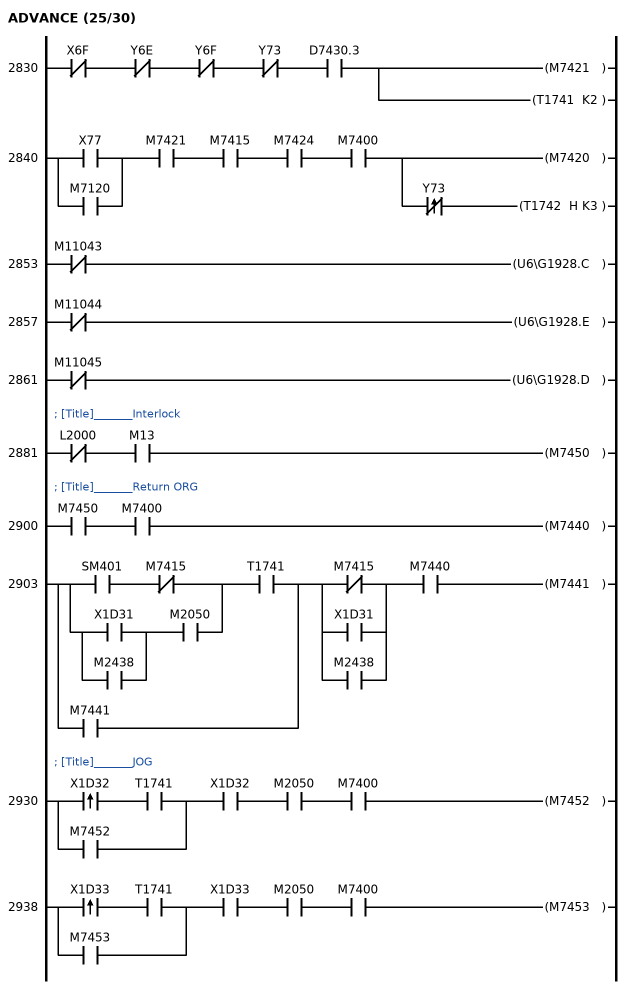
[picture p384: ladder of ADVANCE, rungs at steps 2830 to 2938]
2830  LDI     X6F
      ANI     Y6E
      ANI     Y6F
      ANI     Y73
      AND     D7430.3
      OUT     M7421
      OUT     T1741 K2
2840  LD      X77
      OR      M7120
      AND     M7421
      AND     M7415
      AND     M7424
      AND     M7400
      OUT     M7420
      ANDPI   Y73
      OUTH    T1742 K3
2853  LDI     M11043
      OUT     U6\G1928.C
2857  LDI     M11044
      OUT     U6\G1928.E
2861  LDI     M11045
      OUT     U6\G1928.D
; 
; [Title]_______Interlock
; 
2881  LDI     L2000
      AND     M13
      OUT     M7450
; 
; [Title]_______Return ORG
; 
2900  LD      M7450
      AND     M7400
      OUT     M7440
2903  LD      SM401
      ANI     M7415
      LD      X1D31
      OR      M2438
      AND     M2050
      ORB
      AND     T1741
      OR      M7441
      LDI     M7415
      OR      X1D31
      OR      M2438
      ANB
      AND     M7440
      OUT     M7441
; 
; [Title]_______JOG
; 
2930  LDP     X1D32
      AND     T1741
      OR      M7452
      AND     X1D32
      AND     M2050
      AND     M7400
      OUT     M7452
2938  LDP     X1D33
      AND     T1741
      OR      M7453
      AND     X1D33
      AND     M2050
      AND     M7400
      OUT     M7453
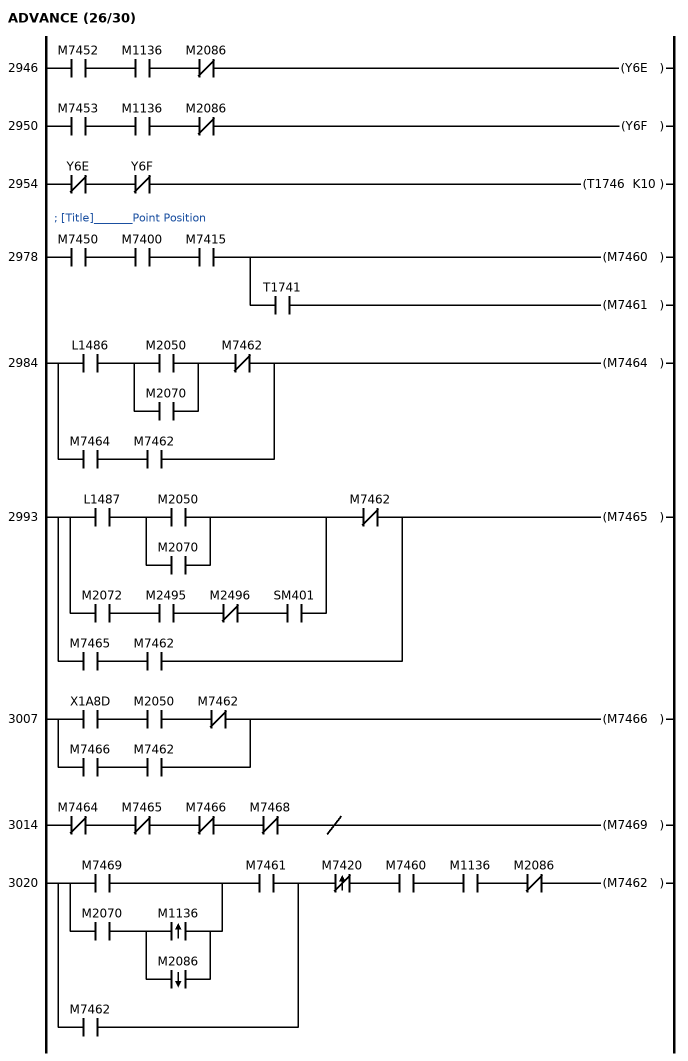
2946  LD      M7452
      AND     M1136
      ANI     M2086
      OUT     Y6E
2950  LD      M7453
      AND     M1136
      ANI     M2086
      OUT     Y6F
2954  LDI     Y6E
      ANI     Y6F
      OUT     T1746 K10
; 
; [Title]_______Point Position
; 
2978  LD      M7450
      AND     M7400
      AND     M7415
      OUT     M7460
      AND     T1741
      OUT     M7461
2984  LD      L1486
      LD      M2050
      OR      M2070
      ANB
      ANI     M7462
      LD      M7464
      AND     M7462
      ORB
      OUT     M7464
2993  LD      L1487
      LD      M2050
      OR      M2070
      ANB
      LD      M2072
      AND     M2495
      ANI     M2496
      AND     SM401
      ORB
      ANI     M7462
      LD      M7465
      AND     M7462
      ORB
      OUT     M7465
3007  LD      X1A8D
      AND     M2050
      ANI     M7462
      LD      M7466
      AND     M7462
      ORB
      OUT     M7466
3014  LDI     M7464
      ANI     M7465
      ANI     M7466
      ANI     M7468
      INV
      OUT     M7469
3020  LD      M7469
      LD      M2070
      LDP     M1136
      ORF     M2086
      ANB
      ORB
      AND     M7461
      OR      M7462
      ANDPI   M7420
      AND     M7460
      AND     M1136
      ANI     M2086
      OUT     M7462
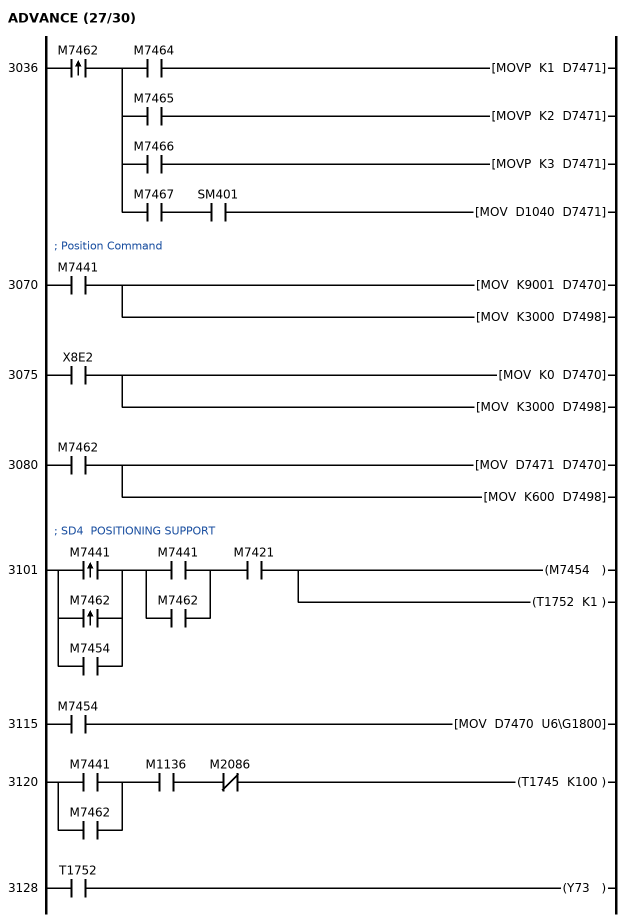
3036  LDP     M7462
      MPS
      AND     M7464
      MOVP    K1 D7471
      MRD
      AND     M7465
      MOVP    K2 D7471
      MRD
      AND     M7466
      MOVP    K3 D7471
      MPP
      AND     M7467
      AND     SM401
      MOV     D1040 D7471
; 
; Position Command
; 
3070  LD      M7441
      MOV     K9001 D7470
      MOV     K3000 D7498
3075  LD      X8E2
      MOV     K0 D7470
      MOV     K3000 D7498
3080  LD      M7462
      MOV     D7471 D7470
      MOV     K600 D7498
; 
; SD4  POSITIONING SUPPORT
; 
3101  LDP     M7441
      ORP     M7462
      OR      M7454
      LD      M7441
      OR      M7462
      ANB
      AND     M7421
      OUT     M7454
      OUT     T1752 K1
3115  LD      M7454
      MOV     D7470 U6\G1800
3120  LD      M7441
      OR      M7462
      AND     M1136
      ANI     M2086
      OUT     T1745 K100
3128  LD      T1752
      OUT     Y73
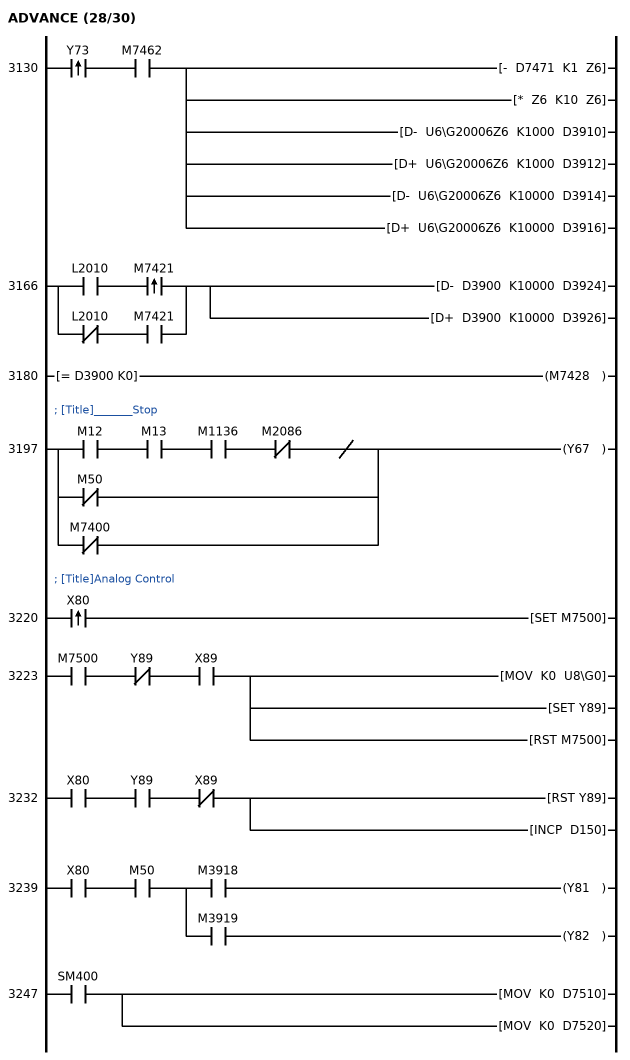
3130  LDP     Y73
      AND     M7462
      -       D7471 K1 Z6
      *       Z6 K10 Z6
      D-      U6\G20006Z6 K1000 D3910
      D+      U6\G20006Z6 K1000 D3912
      D-      U6\G20006Z6 K10000 D3914
      D+      U6\G20006Z6 K10000 D3916
3166  LD      L2010
      ANDP    M7421
      LDI     L2010
      AND     M7421
      ORB
      D-      D3900 K10000 D3924
      D+      D3900 K10000 D3926
3180  LD=     D3900 K0
      OUT     M7428
; 
; [Title]_______Stop
; 
3197  LD      M12
      AND     M13
      AND     M1136
      ANI     M2086
      INV
      ORI     M50
      ORI     M7400
      OUT     Y67
; 
; [Title]Analog Control
; 
3220  LDP     X80
      SET     M7500
3223  LD      M7500
      ANI     Y89
      AND     X89
      MOV     K0 U8\G0
      SET     Y89
      RST     M7500
3232  LD      X80
      AND     Y89
      ANI     X89
      RST     Y89
      INCP    D150
3239  LD      X80
      AND     M50
      MPS
      AND     M3918
      OUT     Y81
      MPP
      AND     M3919
      OUT     Y82
3247  LD      SM400
      MOV     K0 D7510
      MOV     K0 D7520
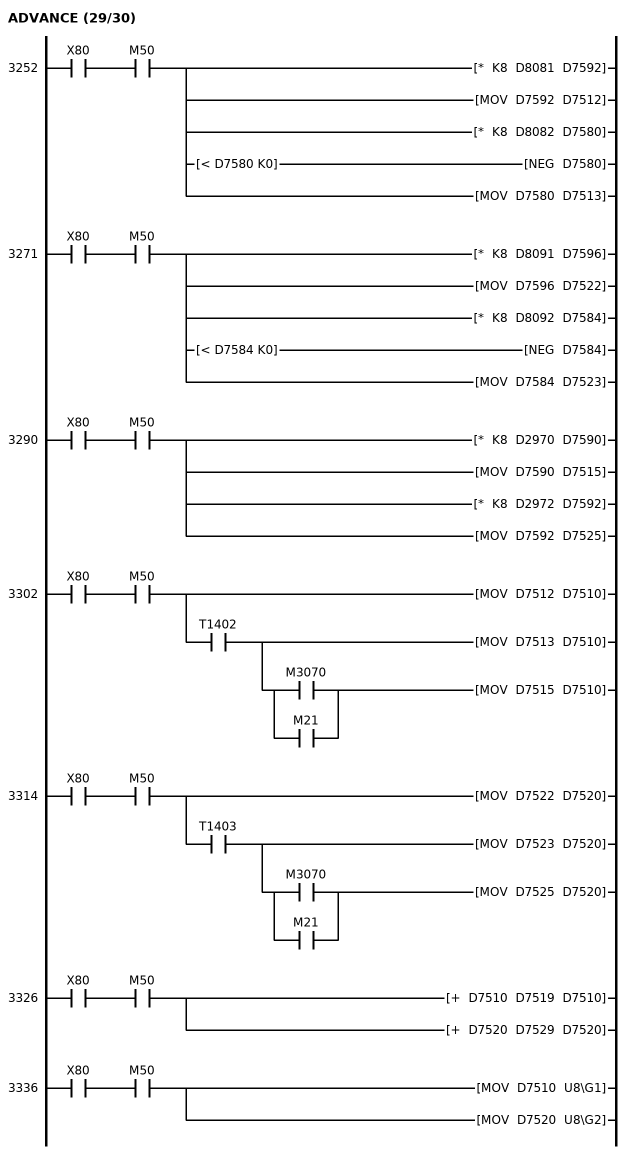
3252  LD      X80
      AND     M50
      *       K8 D8081 D7592
      MOV     D7592 D7512
      *       K8 D8082 D7580
      MPS
      AND<    D7580 K0
      NEG     D7580
      MPP
      MOV     D7580 D7513
3271  LD      X80
      AND     M50
      *       K8 D8091 D7596
      MOV     D7596 D7522
      *       K8 D8092 D7584
      MPS
      AND<    D7584 K0
      NEG     D7584
      MPP
      MOV     D7584 D7523
3290  LD      X80
      AND     M50
      *       K8 D2970 D7590
      MOV     D7590 D7515
      *       K8 D2972 D7592
      MOV     D7592 D7525
3302  LD      X80
      AND     M50
      MOV     D7512 D7510
      AND     T1402
      MOV     D7513 D7510
      LD      M3070
      OR      M21
      ANB
      MOV     D7515 D7510
3314  LD      X80
      AND     M50
      MOV     D7522 D7520
      AND     T1403
      MOV     D7523 D7520
      LD      M3070
      OR      M21
      ANB
      MOV     D7525 D7520
3326  LD      X80
      AND     M50
      +       D7510 D7519 D7510
      +       D7520 D7529 D7520
3336  LD      X80
      AND     M50
      MOV     D7510 U8\G1
      MOV     D7520 U8\G2
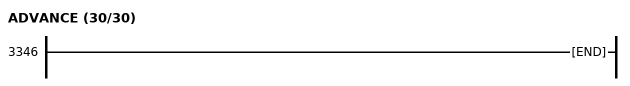
3346  END
END_PROGRAM

PROGRAM ALARM
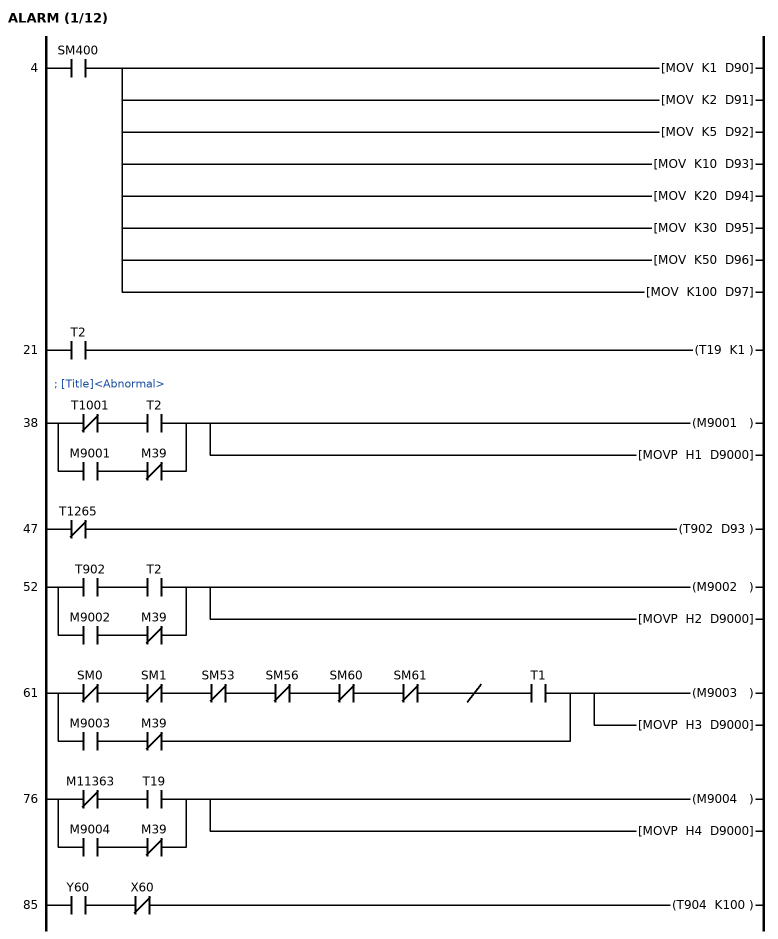
; 
; 
; 
4     LD      SM400
      MOV     K1 D90
      MOV     K2 D91
      MOV     K5 D92
      MOV     K10 D93
      MOV     K20 D94
      MOV     K30 D95
      MOV     K50 D96
      MOV     K100 D97
21    LD      T2
      OUT     T19 K1
; 
; [Title]<Abnormal>
38    LDI     T1001
      AND     T2
      LD      M9001
      ANI     M39
      ORB
      OUT     M9001
      MOVP    H1 D9000
47    LDI     T1265
      OUT     T902 D93
52    LD      T902
      AND     T2
      LD      M9002
      ANI     M39
      ORB
      OUT     M9002
      MOVP    H2 D9000
61    LDI     SM0
      ANI     SM1
      ANI     SM53
      ANI     SM56
      ANI     SM60
      ANI     SM61
      INV
      AND     T1
      LD      M9003
      ANI     M39
      ORB
      OUT     M9003
      MOVP    H3 D9000
76    LDI     M11363
      AND     T19
      LD      M9004
      ANI     M39
      ORB
      OUT     M9004
      MOVP    H4 D9000
85    LD      Y60
      ANI     X60
      OUT     T904 K100
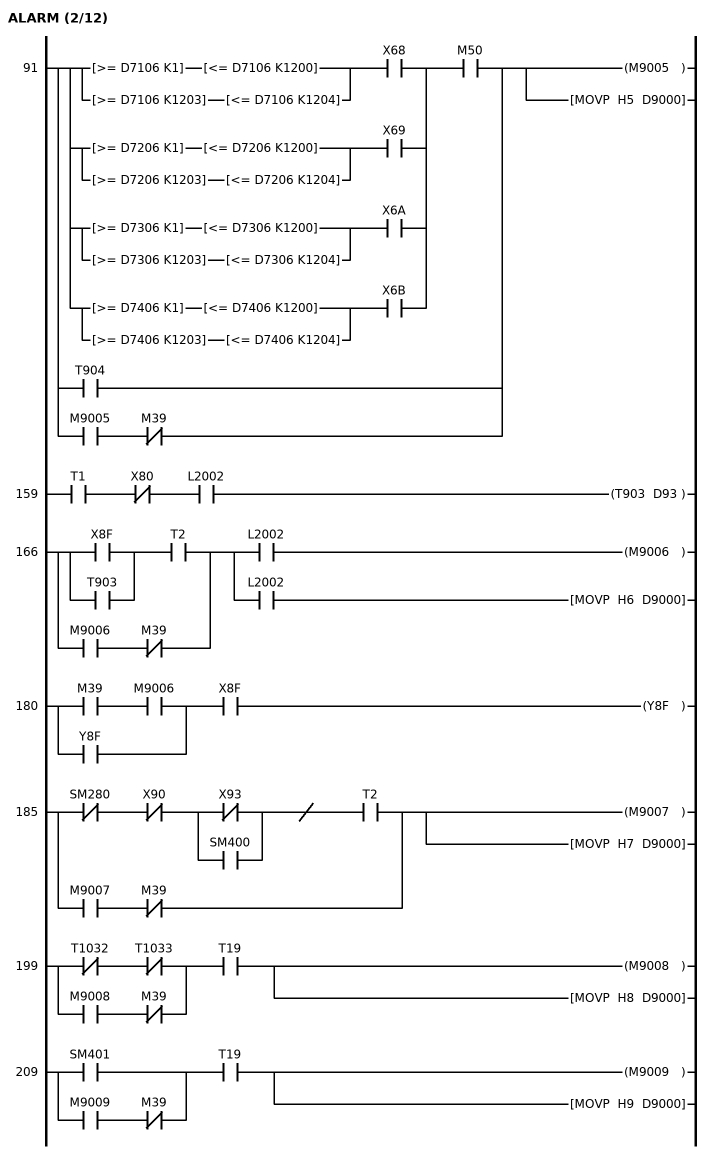
91    LD>=    D7106 K1
      AND<=   D7106 K1200
      LD>=    D7106 K1203
      AND<=   D7106 K1204
      ORB
      AND     X68
      LD>=    D7206 K1
      AND<=   D7206 K1200
      LD>=    D7206 K1203
      AND<=   D7206 K1204
      ORB
      AND     X69
      ORB
      LD>=    D7306 K1
      AND<=   D7306 K1200
      LD>=    D7306 K1203
      AND<=   D7306 K1204
      ORB
      AND     X6A
      ORB
      LD>=    D7406 K1
      AND<=   D7406 K1200
      LD>=    D7406 K1203
      AND<=   D7406 K1204
      ORB
      AND     X6B
      ORB
      AND     M50
      OR      T904
      LD      M9005
      ANI     M39
      ORB
      OUT     M9005
      MOVP    H5 D9000
159   LD      T1
      ANI     X80
      AND     L2002
      OUT     T903 D93
166   LD      X8F
      OR      T903
      AND     T2
      LD      M9006
      ANI     M39
      ORB
      MPS
      AND     L2002
      OUT     M9006
      MPP
      AND     L2002
      MOVP    H6 D9000
180   LD      M39
      AND     M9006
      OR      Y8F
      AND     X8F
      OUT     Y8F
185   LDI     SM280
      ANI     X90
      LDI     X93
      OR      SM400
      ANB
      INV
      AND     T2
      LD      M9007
      ANI     M39
      ORB
      OUT     M9007
      MOVP    H7 D9000
199   LDI     T1032
      ANI     T1033
      LD      M9008
      ANI     M39
      ORB
      AND     T19
      OUT     M9008
      MOVP    H8 D9000
209   LD      SM401
      LD      M9009
      ANI     M39
      ORB
      AND     T19
      OUT     M9009
      MOVP    H9 D9000
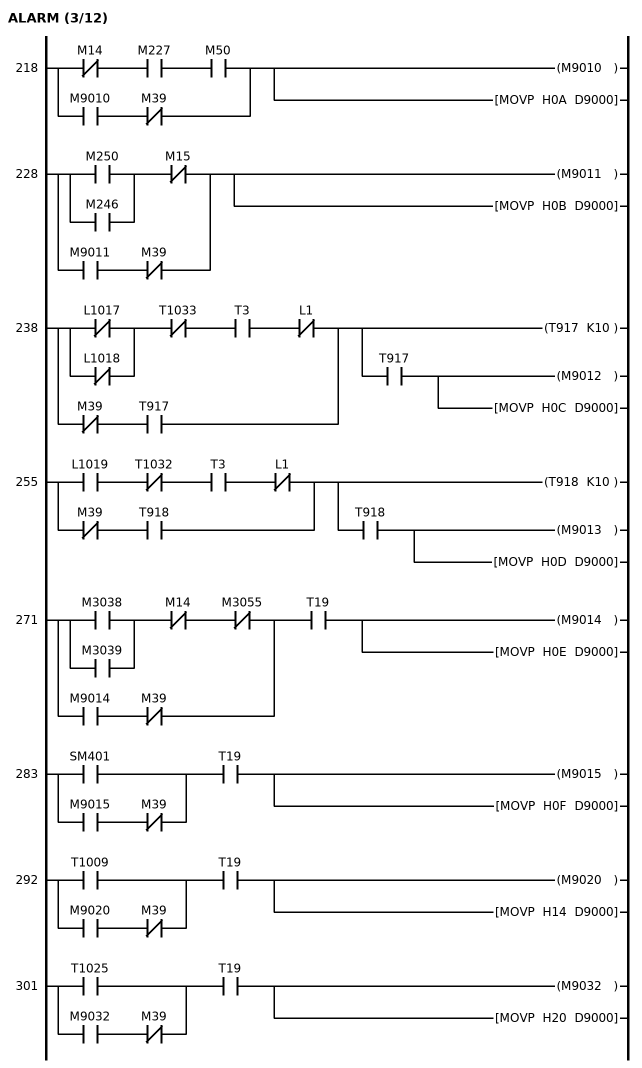
218   LDI     M14
      AND     M227
      AND     M50
      LD      M9010
      ANI     M39
      ORB
      OUT     M9010
      MOVP    H0A D9000
228   LD      M250
      OR      M246
      ANI     M15
      LD      M9011
      ANI     M39
      ORB
      OUT     M9011
      MOVP    H0B D9000
238   LDI     L1017
      ORI     L1018
      ANI     T1033
      AND     T3
      ANI     L1
      LDI     M39
      AND     T917
      ORB
      OUT     T917 K10
      AND     T917
      OUT     M9012
      MOVP    H0C D9000
255   LD      L1019
      ANI     T1032
      AND     T3
      ANI     L1
      LDI     M39
      AND     T918
      ORB
      OUT     T918 K10
      AND     T918
      OUT     M9013
      MOVP    H0D D9000
271   LD      M3038
      OR      M3039
      ANI     M14
      ANI     M3055
      LD      M9014
      ANI     M39
      ORB
      AND     T19
      OUT     M9014
      MOVP    H0E D9000
283   LD      SM401
      LD      M9015
      ANI     M39
      ORB
      AND     T19
      OUT     M9015
      MOVP    H0F D9000
292   LD      T1009
      LD      M9020
      ANI     M39
      ORB
      AND     T19
      OUT     M9020
      MOVP    H14 D9000
301   LD      T1025
      LD      M9032
      ANI     M39
      ORB
      AND     T19
      OUT     M9032
      MOVP    H20 D9000
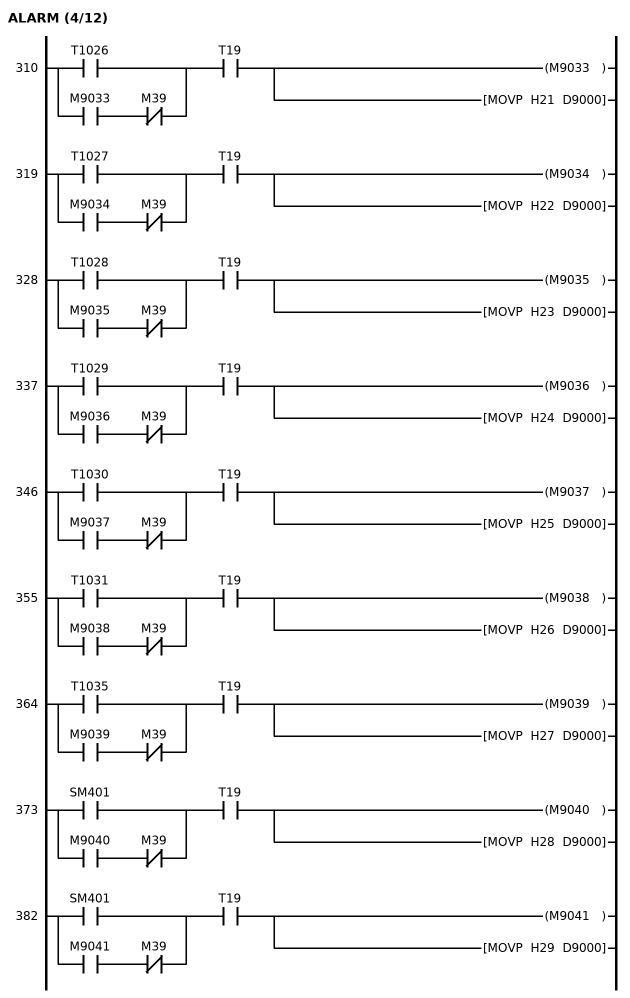
310   LD      T1026
      LD      M9033
      ANI     M39
      ORB
      AND     T19
      OUT     M9033
      MOVP    H21 D9000
319   LD      T1027
      LD      M9034
      ANI     M39
      ORB
      AND     T19
      OUT     M9034
      MOVP    H22 D9000
328   LD      T1028
      LD      M9035
      ANI     M39
      ORB
      AND     T19
      OUT     M9035
      MOVP    H23 D9000
337   LD      T1029
      LD      M9036
      ANI     M39
      ORB
      AND     T19
      OUT     M9036
      MOVP    H24 D9000
346   LD      T1030
      LD      M9037
      ANI     M39
      ORB
      AND     T19
      OUT     M9037
      MOVP    H25 D9000
355   LD      T1031
      LD      M9038
      ANI     M39
      ORB
      AND     T19
      OUT     M9038
      MOVP    H26 D9000
364   LD      T1035
      LD      M9039
      ANI     M39
      ORB
      AND     T19
      OUT     M9039
      MOVP    H27 D9000
373   LD      SM401
      LD      M9040
      ANI     M39
      ORB
      AND     T19
      OUT     M9040
      MOVP    H28 D9000
382   LD      SM401
      LD      M9041
      ANI     M39
      ORB
      AND     T19
      OUT     M9041
      MOVP    H29 D9000
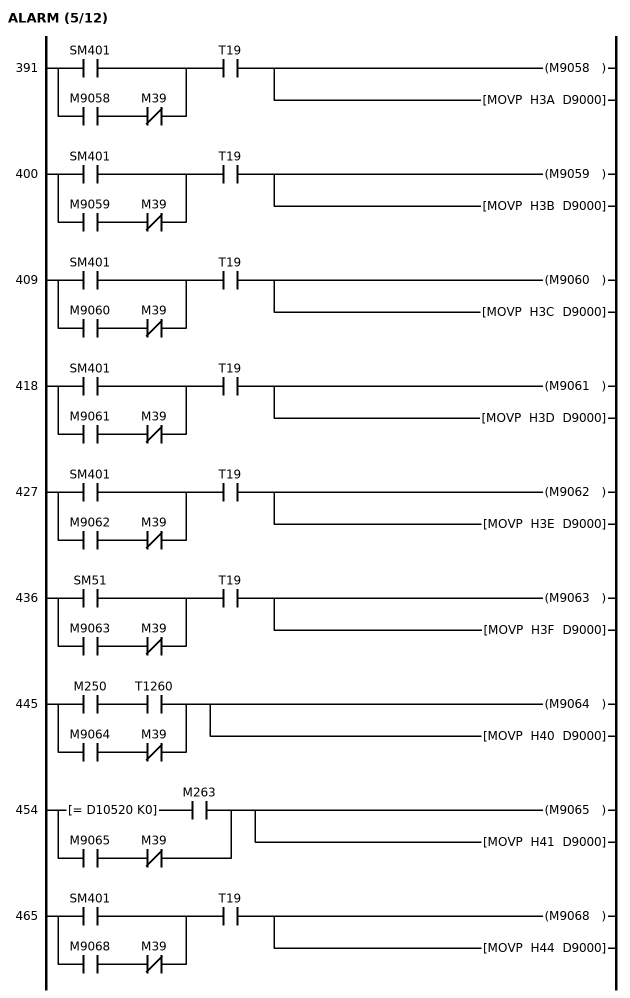
391   LD      SM401
      LD      M9058
      ANI     M39
      ORB
      AND     T19
      OUT     M9058
      MOVP    H3A D9000
400   LD      SM401
      LD      M9059
      ANI     M39
      ORB
      AND     T19
      OUT     M9059
      MOVP    H3B D9000
409   LD      SM401
      LD      M9060
      ANI     M39
      ORB
      AND     T19
      OUT     M9060
      MOVP    H3C D9000
418   LD      SM401
      LD      M9061
      ANI     M39
      ORB
      AND     T19
      OUT     M9061
      MOVP    H3D D9000
427   LD      SM401
      LD      M9062
      ANI     M39
      ORB
      AND     T19
      OUT     M9062
      MOVP    H3E D9000
436   LD      SM51
      LD      M9063
      ANI     M39
      ORB
      AND     T19
      OUT     M9063
      MOVP    H3F D9000
445   LD      M250
      AND     T1260
      LD      M9064
      ANI     M39
      ORB
      OUT     M9064
      MOVP    H40 D9000
454   LD=     D10520 K0
      AND     M263
      LD      M9065
      ANI     M39
      ORB
      OUT     M9065
      MOVP    H41 D9000
465   LD      SM401
      LD      M9068
      ANI     M39
      ORB
      AND     T19
      OUT     M9068
      MOVP    H44 D9000
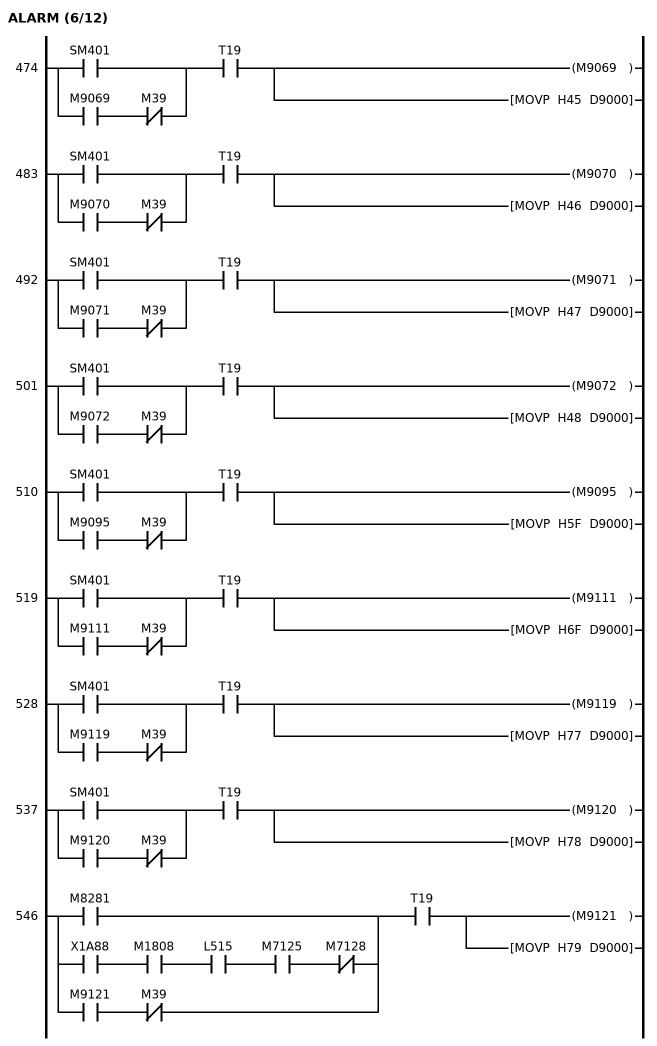
474   LD      SM401
      LD      M9069
      ANI     M39
      ORB
      AND     T19
      OUT     M9069
      MOVP    H45 D9000
483   LD      SM401
      LD      M9070
      ANI     M39
      ORB
      AND     T19
      OUT     M9070
      MOVP    H46 D9000
492   LD      SM401
      LD      M9071
      ANI     M39
      ORB
      AND     T19
      OUT     M9071
      MOVP    H47 D9000
501   LD      SM401
      LD      M9072
      ANI     M39
      ORB
      AND     T19
      OUT     M9072
      MOVP    H48 D9000
510   LD      SM401
      LD      M9095
      ANI     M39
      ORB
      AND     T19
      OUT     M9095
      MOVP    H5F D9000
519   LD      SM401
      LD      M9111
      ANI     M39
      ORB
      AND     T19
      OUT     M9111
      MOVP    H6F D9000
528   LD      SM401
      LD      M9119
      ANI     M39
      ORB
      AND     T19
      OUT     M9119
      MOVP    H77 D9000
537   LD      SM401
      LD      M9120
      ANI     M39
      ORB
      AND     T19
      OUT     M9120
      MOVP    H78 D9000
546   LD      M8281
      LD      X1A88
      AND     M1808
      AND     L515
      AND     M7125
      ANI     M7128
      ORB
      LD      M9121
      ANI     M39
      ORB
      AND     T19
      OUT     M9121
      MOVP    H79 D9000
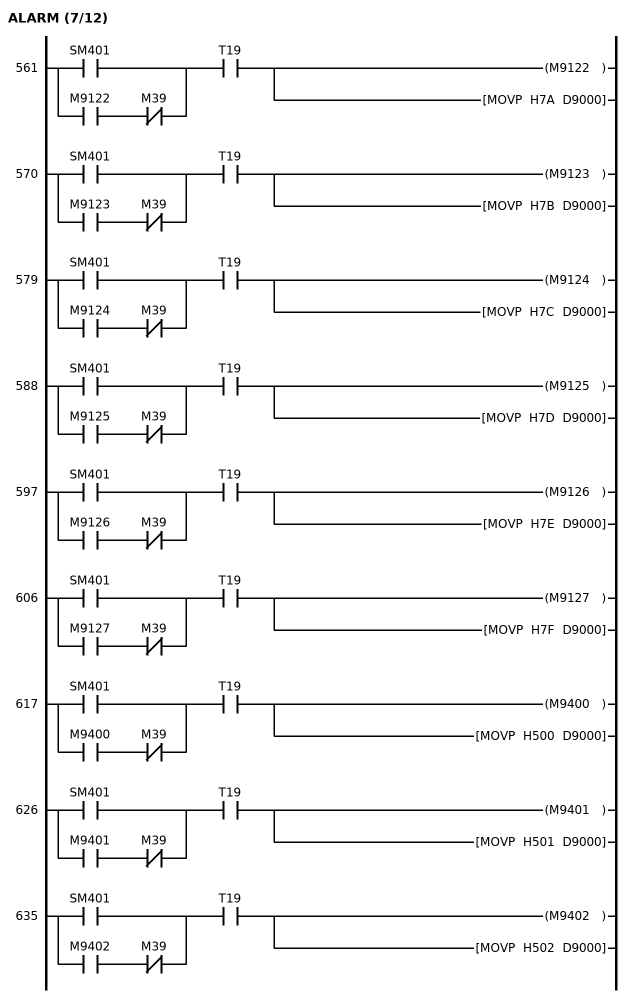
561   LD      SM401
      LD      M9122
      ANI     M39
      ORB
      AND     T19
      OUT     M9122
      MOVP    H7A D9000
570   LD      SM401
      LD      M9123
      ANI     M39
      ORB
      AND     T19
      OUT     M9123
      MOVP    H7B D9000
579   LD      SM401
      LD      M9124
      ANI     M39
      ORB
      AND     T19
      OUT     M9124
      MOVP    H7C D9000
588   LD      SM401
      LD      M9125
      ANI     M39
      ORB
      AND     T19
      OUT     M9125
      MOVP    H7D D9000
597   LD      SM401
      LD      M9126
      ANI     M39
      ORB
      AND     T19
      OUT     M9126
      MOVP    H7E D9000
606   LD      SM401
      LD      M9127
      ANI     M39
      ORB
      AND     T19
      OUT     M9127
      MOVP    H7F D9000
; 
; 
617   LD      SM401
      LD      M9400
      ANI     M39
      ORB
      AND     T19
      OUT     M9400
      MOVP    H500 D9000
626   LD      SM401
      LD      M9401
      ANI     M39
      ORB
      AND     T19
      OUT     M9401
      MOVP    H501 D9000
635   LD      SM401
      LD      M9402
      ANI     M39
      ORB
      AND     T19
      OUT     M9402
      MOVP    H502 D9000
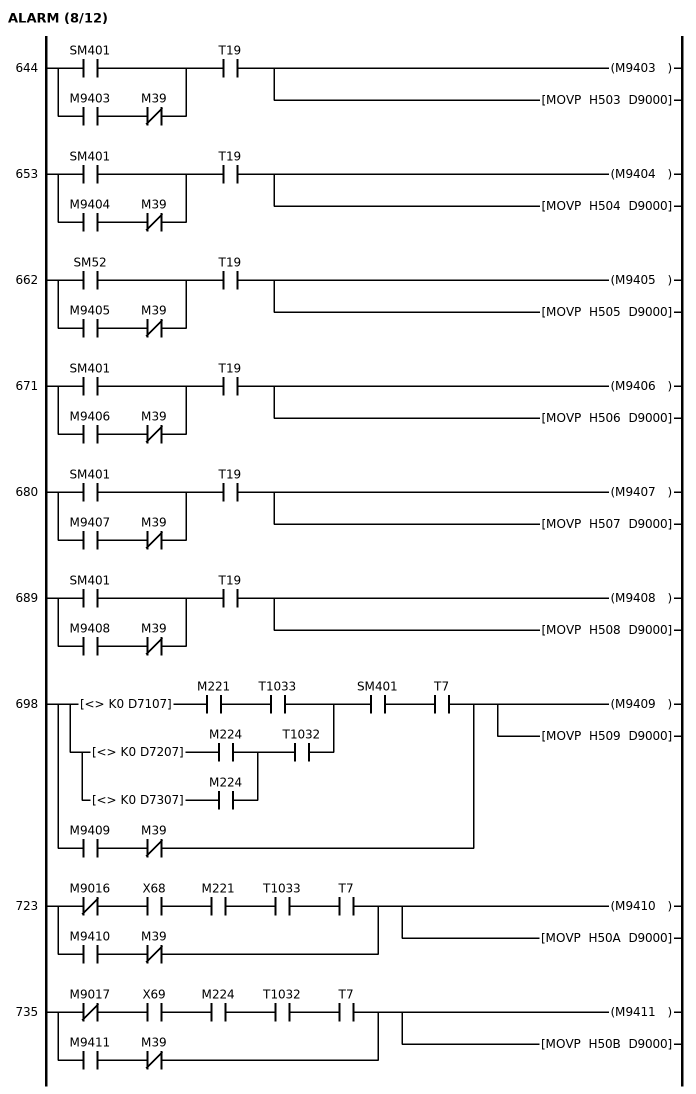
644   LD      SM401
      LD      M9403
      ANI     M39
      ORB
      AND     T19
      OUT     M9403
      MOVP    H503 D9000
653   LD      SM401
      LD      M9404
      ANI     M39
      ORB
      AND     T19
      OUT     M9404
      MOVP    H504 D9000
662   LD      SM52
      LD      M9405
      ANI     M39
      ORB
      AND     T19
      OUT     M9405
      MOVP    H505 D9000
671   LD      SM401
      LD      M9406
      ANI     M39
      ORB
      AND     T19
      OUT     M9406
      MOVP    H506 D9000
680   LD      SM401
      LD      M9407
      ANI     M39
      ORB
      AND     T19
      OUT     M9407
      MOVP    H507 D9000
689   LD      SM401
      LD      M9408
      ANI     M39
      ORB
      AND     T19
      OUT     M9408
      MOVP    H508 D9000
698   LD<>    K0 D7107
      AND     M221
      AND     T1033
      LD<>    K0 D7207
      AND     M224
      LD<>    K0 D7307
      AND     M224
      ORB
      AND     T1032
      ORB
      AND     SM401
      AND     T7
      LD      M9409
      ANI     M39
      ORB
      OUT     M9409
      MOVP    H509 D9000
723   LDI     M9016
      AND     X68
      AND     M221
      AND     T1033
      AND     T7
      LD      M9410
      ANI     M39
      ORB
      OUT     M9410
      MOVP    H50A D9000
735   LDI     M9017
      AND     X69
      AND     M224
      AND     T1032
      AND     T7
      LD      M9411
      ANI     M39
      ORB
      OUT     M9411
      MOVP    H50B D9000
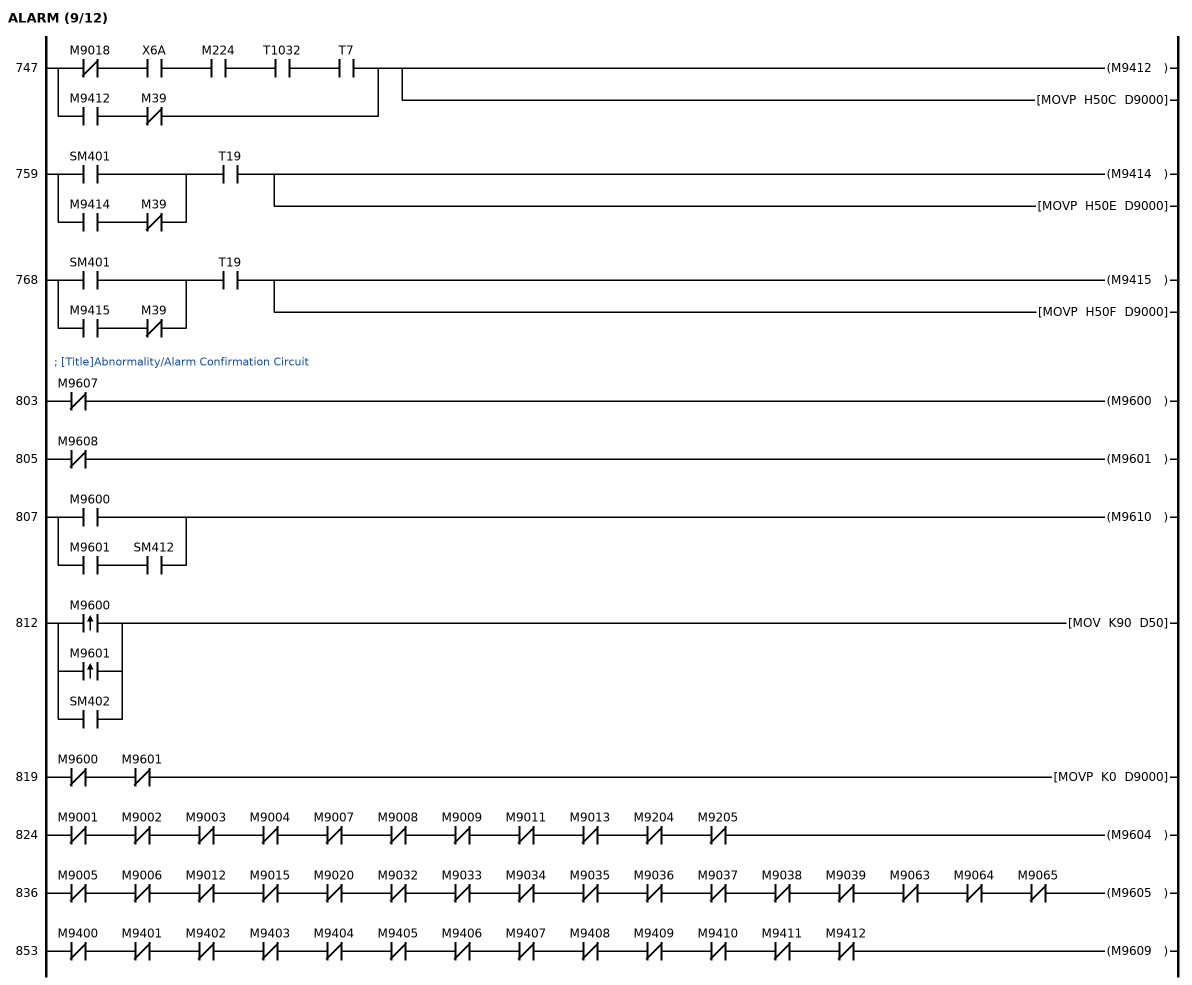
747   LDI     M9018
      AND     X6A
      AND     M224
      AND     T1032
      AND     T7
      LD      M9412
      ANI     M39
      ORB
      OUT     M9412
      MOVP    H50C D9000
759   LD      SM401
      LD      M9414
      ANI     M39
      ORB
      AND     T19
      OUT     M9414
      MOVP    H50E D9000
768   LD      SM401
      LD      M9415
      ANI     M39
      ORB
      AND     T19
      OUT     M9415
      MOVP    H50F D9000
; 
; [Title]Abnormality/Alarm Confirmation Circuit
803   LDI     M9607
      OUT     M9600
805   LDI     M9608
      OUT     M9601
807   LD      M9600
      LD      M9601
      AND     SM412
      ORB
      OUT     M9610
812   LDP     M9600
      ORP     M9601
      OR      SM402
      MOV     K90 D50
819   LDI     M9600
      ANI     M9601
      MOVP    K0 D9000
824   LDI     M9001
      ANI     M9002
      ANI     M9003
      ANI     M9004
      ANI     M9007
      ANI     M9008
      ANI     M9009
      ANI     M9011
      ANI     M9013
      ANI     M9204
      ANI     M9205
      OUT     M9604
836   LDI     M9005
      ANI     M9006
      ANI     M9012
      ANI     M9015
      ANI     M9020
      ANI     M9032
      ANI     M9033
      ANI     M9034
      ANI     M9035
      ANI     M9036
      ANI     M9037
      ANI     M9038
      ANI     M9039
      ANI     M9063
      ANI     M9064
      ANI     M9065
      OUT     M9605
853   LDI     M9400
      ANI     M9401
      ANI     M9402
      ANI     M9403
      ANI     M9404
      ANI     M9405
      ANI     M9406
      ANI     M9407
      ANI     M9408
      ANI     M9409
      ANI     M9410
      ANI     M9411
      ANI     M9412
      OUT     M9609
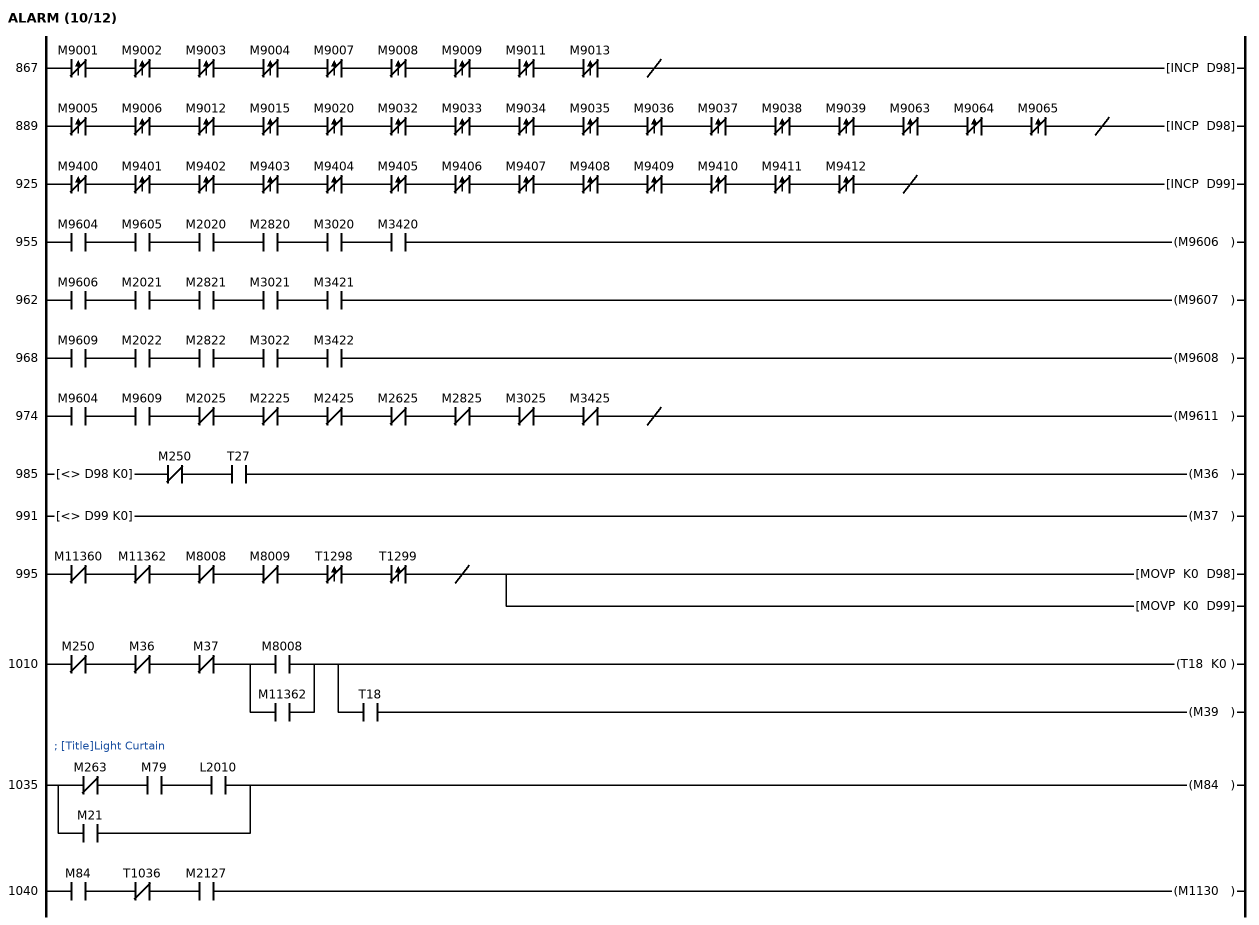
867   LDPI    M9001
      ANDPI   M9002
      ANDPI   M9003
      ANDPI   M9004
      ANDPI   M9007
      ANDPI   M9008
      ANDPI   M9009
      ANDPI   M9011
      ANDPI   M9013
      INV
      INCP    D98
889   LDPI    M9005
      ANDPI   M9006
      ANDPI   M9012
      ANDPI   M9015
      ANDPI   M9020
      ANDPI   M9032
      ANDPI   M9033
      ANDPI   M9034
      ANDPI   M9035
      ANDPI   M9036
      ANDPI   M9037
      ANDPI   M9038
      ANDPI   M9039
      ANDPI   M9063
      ANDPI   M9064
      ANDPI   M9065
      INV
      INCP    D98
925   LDPI    M9400
      ANDPI   M9401
      ANDPI   M9402
      ANDPI   M9403
      ANDPI   M9404
      ANDPI   M9405
      ANDPI   M9406
      ANDPI   M9407
      ANDPI   M9408
      ANDPI   M9409
      ANDPI   M9410
      ANDPI   M9411
      ANDPI   M9412
      INV
      INCP    D99
955   LD      M9604
      AND     M9605
      AND     M2020
      AND     M2820
      AND     M3020
      AND     M3420
      OUT     M9606
962   LD      M9606
      AND     M2021
      AND     M2821
      AND     M3021
      AND     M3421
      OUT     M9607
968   LD      M9609
      AND     M2022
      AND     M2822
      AND     M3022
      AND     M3422
      OUT     M9608
974   LD      M9604
      AND     M9609
      ANI     M2025
      ANI     M2225
      ANI     M2425
      ANI     M2625
      ANI     M2825
      ANI     M3025
      ANI     M3425
      INV
      OUT     M9611
985   LD<>    D98 K0
      ANI     M250
      AND     T27
      OUT     M36
991   LD<>    D99 K0
      OUT     M37
995   LDI     M11360
      ANI     M11362
      ANI     M8008
      ANI     M8009
      ANDPI   T1298
      ANDPI   T1299
      INV
      MOVP    K0 D98
      MOVP    K0 D99
1010  LDI     M250
      ANI     M36
      ANI     M37
      LD      M8008
      OR      M11362
      ANB
      OUT     T18 K0
      AND     T18
      OUT     M39
; [Title]Light Curtain
; 
1035  LDI     M263
      AND     M79
      AND     L2010
      OR      M21
      OUT     M84
1040  LD      M84
      ANI     T1036
      AND     M2127
      OUT     M1130
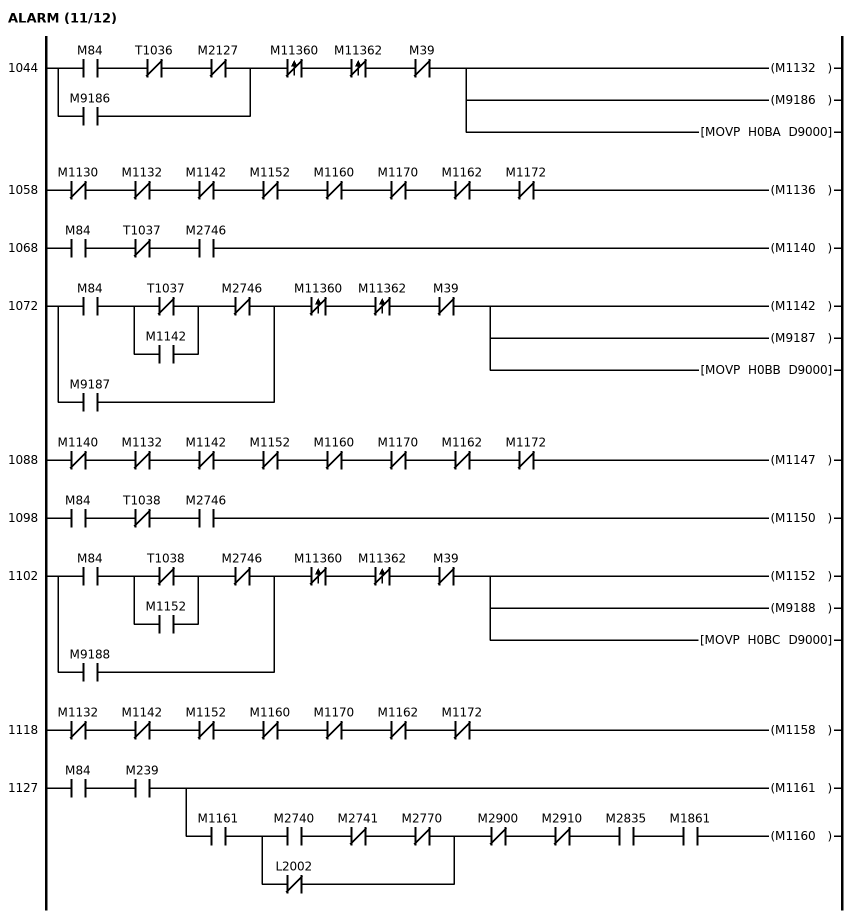
1044  LD      M84
      ANI     T1036
      ANI     M2127
      OR      M9186
      ANDPI   M11360
      ANDPI   M11362
      ANI     M39
      OUT     M1132
      OUT     M9186
      MOVP    H0BA D9000
1058  LDI     M1130
      ANI     M1132
      ANI     M1142
      ANI     M1152
      ANI     M1160
      ANI     M1170
      ANI     M1162
      ANI     M1172
      OUT     M1136
; 
1068  LD      M84
      ANI     T1037
      AND     M2746
      OUT     M1140
1072  LD      M84
      LDI     T1037
      OR      M1142
      ANB
      ANI     M2746
      OR      M9187
      ANDPI   M11360
      ANDPI   M11362
      ANI     M39
      OUT     M1142
      OUT     M9187
      MOVP    H0BB D9000
1088  LDI     M1140
      ANI     M1132
      ANI     M1142
      ANI     M1152
      ANI     M1160
      ANI     M1170
      ANI     M1162
      ANI     M1172
      OUT     M1147
; 
1098  LD      M84
      ANI     T1038
      AND     M2746
      OUT     M1150
1102  LD      M84
      LDI     T1038
      OR      M1152
      ANB
      ANI     M2746
      OR      M9188
      ANDPI   M11360
      ANDPI   M11362
      ANI     M39
      OUT     M1152
      OUT     M9188
      MOVP    H0BC D9000
1118  LDI     M1132
      ANI     M1142
      ANI     M1152
      ANI     M1160
      ANI     M1170
      ANI     M1162
      ANI     M1172
      OUT     M1158
; 
1127  LD      M84
      AND     M239
      OUT     M1161
      AND     M1161
      LD      M2740
      ANI     M2741
      ANI     M2770
      ORI     L2002
      ANB
      ANI     M2900
      ANI     M2910
      AND     M2835
      AND     M1861
      OUT     M1160
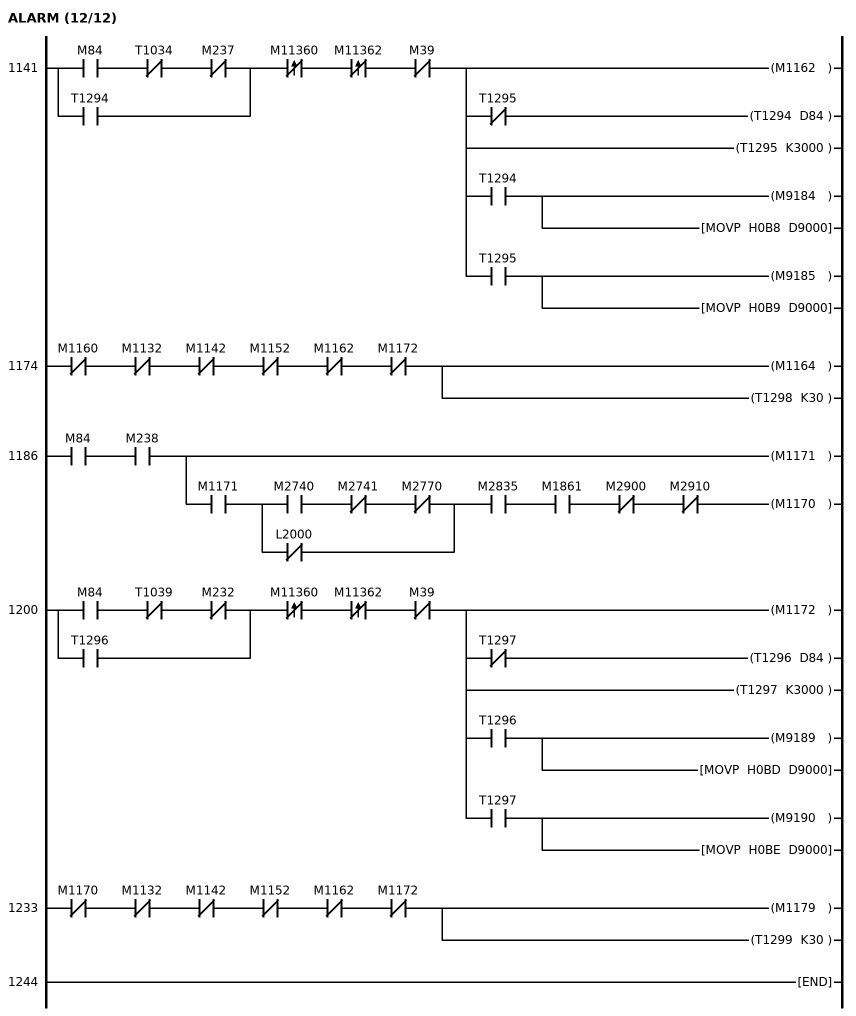
1141  LD      M84
      ANI     T1034
      ANI     M237
      OR      T1294
      ANDPI   M11360
      ANDPI   M11362
      ANI     M39
      OUT     M1162
      MPS
      ANI     T1295
      OUT     T1294 D84
      MPP
      OUT     T1295 K3000
      MPS
      AND     T1294
      OUT     M9184
      MOVP    H0B8 D9000
      MPP
      AND     T1295
      OUT     M9185
      MOVP    H0B9 D9000
1174  LDI     M1160
      ANI     M1132
      ANI     M1142
      ANI     M1152
      ANI     M1162
      ANI     M1172
      OUT     M1164
      OUT     T1298 K30
; 
1186  LD      M84
      AND     M238
      OUT     M1171
      AND     M1171
      LD      M2740
      ANI     M2741
      ANI     M2770
      ORI     L2000
      ANB
      AND     M2835
      AND     M1861
      ANI     M2900
      ANI     M2910
      OUT     M1170
1200  LD      M84
      ANI     T1039
      ANI     M232
      OR      T1296
      ANDPI   M11360
      ANDPI   M11362
      ANI     M39
      OUT     M1172
      MPS
      ANI     T1297
      OUT     T1296 D84
      MPP
      OUT     T1297 K3000
      MPS
      AND     T1296
      OUT     M9189
      MOVP    H0BD D9000
      MPP
      AND     T1297
      OUT     M9190
      MOVP    H0BE D9000
1233  LDI     M1170
      ANI     M1132
      ANI     M1142
      ANI     M1152
      ANI     M1162
      ANI     M1172
      OUT     M1179
      OUT     T1299 K30
1244  END
END_PROGRAM

PROGRAM HMI-TPL
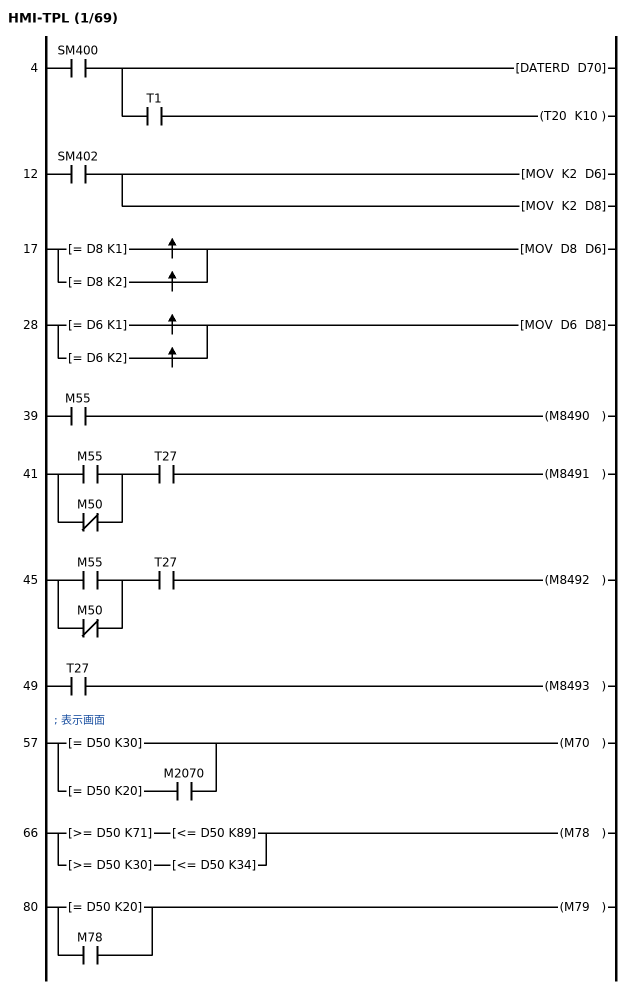
; 
; 
; 
4     LD      SM400
      DATERD  D70
      AND     T1
      OUT     T20 K10
12    LD      SM402
      MOV     K2 D6
      MOV     K2 D8
17    LD=     D8 K1
      MEP
      LD=     D8 K2
      MEP
      ORB
      MOV     D8 D6
28    LD=     D6 K1
      MEP
      LD=     D6 K2
      MEP
      ORB
      MOV     D6 D8
39    LD      M55
      OUT     M8490
41    LD      M55
      ORI     M50
      AND     T27
      OUT     M8491
45    LD      M55
      ORI     M50
      AND     T27
      OUT     M8492
49    LD      T27
      OUT     M8493
; 表示画面
57    LD=     D50 K30
      LD=     D50 K20
      AND     M2070
      ORB
      OUT     M70
66    LD>=    D50 K71
      AND<=   D50 K89
      LD>=    D50 K30
      AND<=   D50 K34
      ORB
      OUT     M78
80    LD=     D50 K20
      OR      M78
      OUT     M79
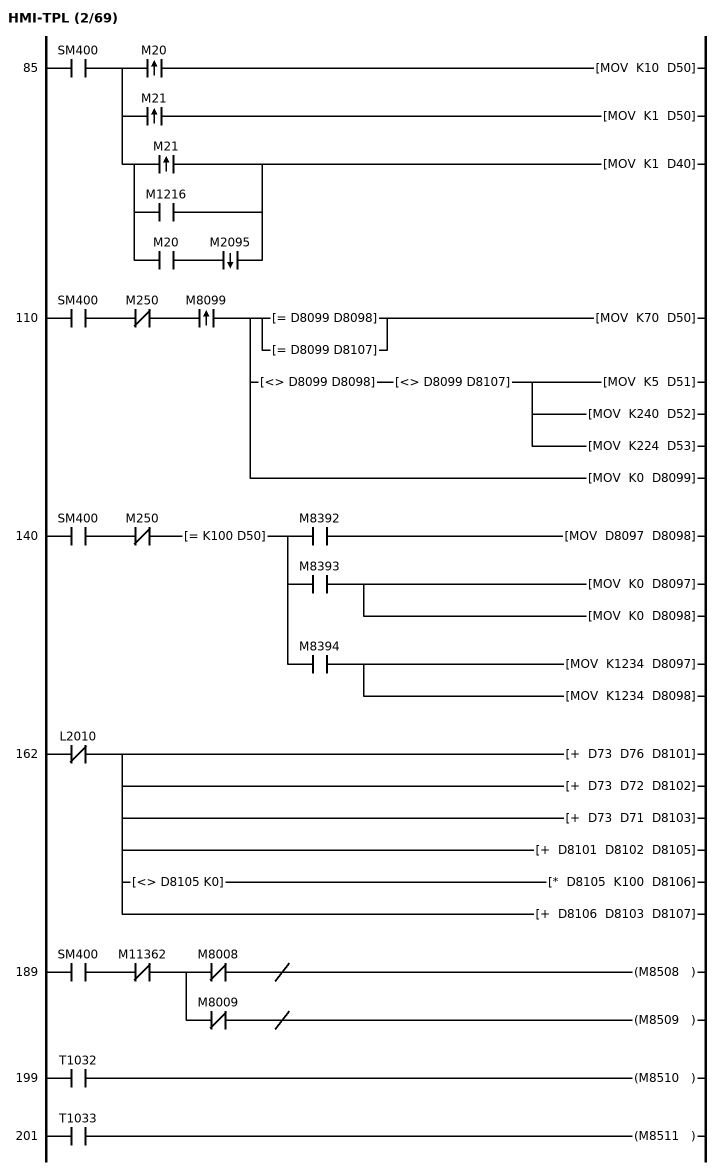
85    LD      SM400
      MPS
      ANDP    M20
      MOV     K10 D50
      MRD
      ANDP    M21
      MOV     K1 D50
      MPP
      LDP     M21
      OR      M1216
      LD      M20
      ANDF    M2095
      ORB
      ANB
      MOV     K1 D40
; 
; 
; 
110   LD      SM400
      ANI     M250
      ANDP    M8099
      MPS
      LD=     D8099 D8098
      OR=     D8099 D8107
      ANB
      MOV     K70 D50
      MRD
      AND<>   D8099 D8098
      AND<>   D8099 D8107
      MOV     K5 D51
      MOV     K240 D52
      MOV     K224 D53
      MPP
      MOV     K0 D8099
140   LD      SM400
      ANI     M250
      AND=    K100 D50
      MPS
      AND     M8392
      MOV     D8097 D8098
      MRD
      AND     M8393
      MOV     K0 D8097
      MOV     K0 D8098
      MPP
      AND     M8394
      MOV     K1234 D8097
      MOV     K1234 D8098
; 
162   LDI     L2010
      +       D73 D76 D8101
      +       D73 D72 D8102
      +       D73 D71 D8103
      +       D8101 D8102 D8105
      MPS
      AND<>   D8105 K0
      *       D8105 K100 D8106
      MPP
      +       D8106 D8103 D8107
; 
; 
; 
189   LD      SM400
      ANI     M11362
      MPS
      ANI     M8008
      INV
      OUT     M8508
      MPP
      ANI     M8009
      INV
      OUT     M8509
199   LD      T1032
      OUT     M8510
201   LD      T1033
      OUT     M8511
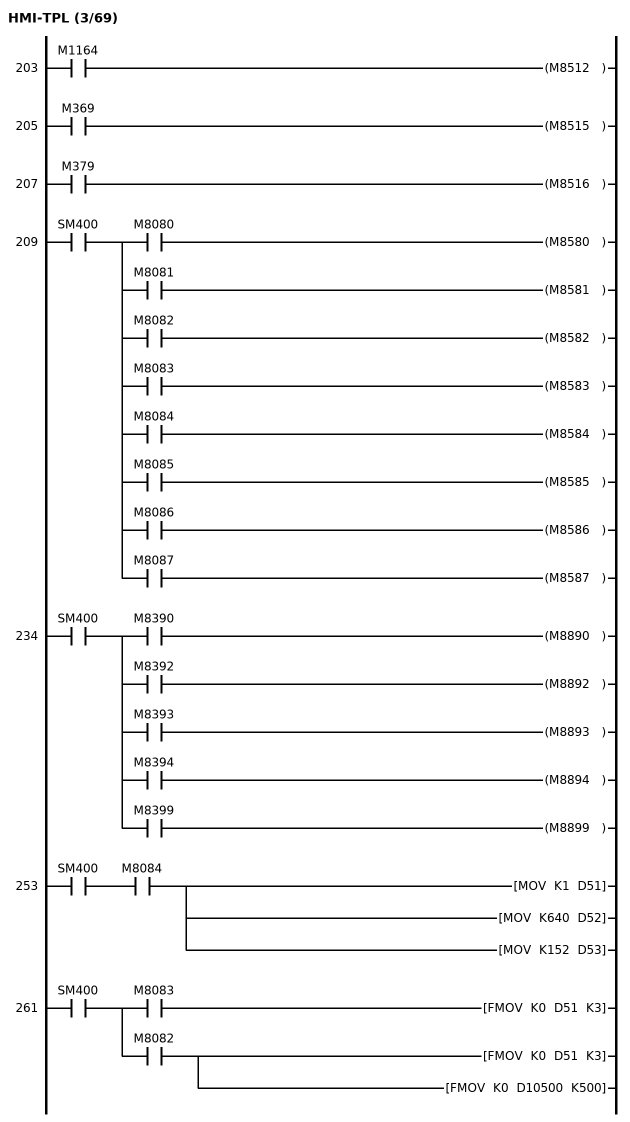
203   LD      M1164
      OUT     M8512
205   LD      M369
      OUT     M8515
207   LD      M379
      OUT     M8516
209   LD      SM400
      MPS
      AND     M8080
      OUT     M8580
      MRD
      AND     M8081
      OUT     M8581
      MRD
      AND     M8082
      OUT     M8582
      MRD
      AND     M8083
      OUT     M8583
      MRD
      AND     M8084
      OUT     M8584
      MRD
      AND     M8085
      OUT     M8585
      MRD
      AND     M8086
      OUT     M8586
      MPP
      AND     M8087
      OUT     M8587
234   LD      SM400
      MPS
      AND     M8390
      OUT     M8890
      MRD
      AND     M8392
      OUT     M8892
      MRD
      AND     M8393
      OUT     M8893
      MRD
      AND     M8394
      OUT     M8894
      MPP
      AND     M8399
      OUT     M8899
; 
; 
; 
253   LD      SM400
      AND     M8084
      MOV     K1 D51
      MOV     K640 D52
      MOV     K152 D53
261   LD      SM400
      MPS
      AND     M8083
      FMOV    K0 D51 K3
      MPP
      AND     M8082
      FMOV    K0 D51 K3
      FMOV    K0 D10500 K500
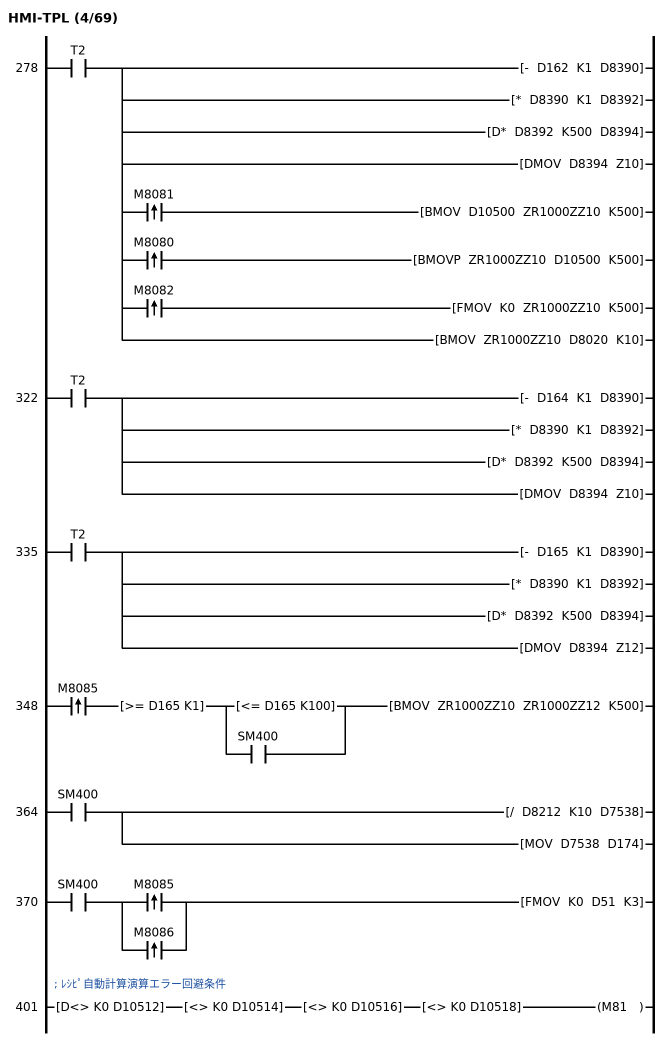
278   LD      T2
      -       D162 K1 D8390
      *       D8390 K1 D8392
      D*      D8392 K500 D8394
      DMOV    D8394 Z10
      MPS
      ANDP    M8081
      BMOV    D10500 ZR1000ZZ10 K500
      MRD
      ANDP    M8080
      BMOVP   ZR1000ZZ10 D10500 K500
      MRD
      ANDP    M8082
      FMOV    K0 ZR1000ZZ10 K500
      MPP
      BMOV    ZR1000ZZ10 D8020 K10
322   LD      T2
      -       D164 K1 D8390
      *       D8390 K1 D8392
      D*      D8392 K500 D8394
      DMOV    D8394 Z10
335   LD      T2
      -       D165 K1 D8390
      *       D8390 K1 D8392
      D*      D8392 K500 D8394
      DMOV    D8394 Z12
348   LDP     M8085
      AND>=   D165 K1
      LD<=    D165 K100
      OR      SM400
      ANB
      BMOV    ZR1000ZZ10 ZR1000ZZ12 K500
364   LD      SM400
      /       D8212 K10 D7538
      MOV     D7538 D174
370   LD      SM400
      LDP     M8085
      ORP     M8086
      ANB
      FMOV    K0 D51 K3
; 
; 
; 
; ﾚｼﾋﾟ自動計算演算エラー回避条件
401   LDD<>   K0 D10512
      AND<>   K0 D10514
      AND<>   K0 D10516
      AND<>   K0 D10518
      OUT     M81
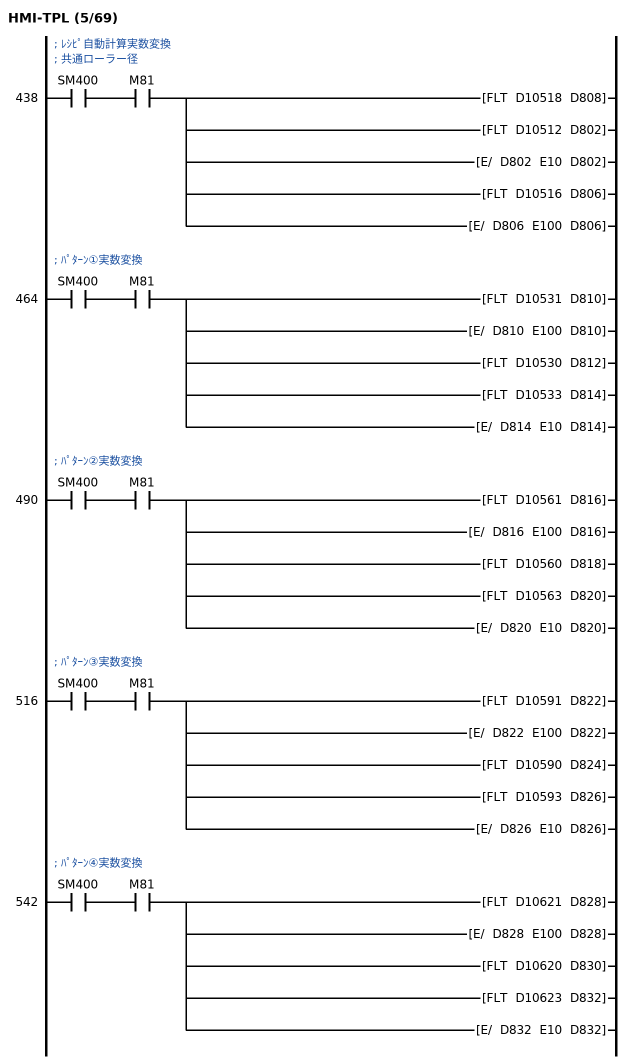
; ﾚｼﾋﾟ自動計算実数変換
; 共通ローラー径
438   LD      SM400
      AND     M81
      FLT     D10518 D808
      FLT     D10512 D802
      E/      D802 E10 D802
      FLT     D10516 D806
      E/      D806 E100 D806
; ﾊﾟﾀｰﾝ①実数変換
464   LD      SM400
      AND     M81
      FLT     D10531 D810
      E/      D810 E100 D810
      FLT     D10530 D812
      FLT     D10533 D814
      E/      D814 E10 D814
; ﾊﾟﾀｰﾝ②実数変換
490   LD      SM400
      AND     M81
      FLT     D10561 D816
      E/      D816 E100 D816
      FLT     D10560 D818
      FLT     D10563 D820
      E/      D820 E10 D820
; ﾊﾟﾀｰﾝ③実数変換
516   LD      SM400
      AND     M81
      FLT     D10591 D822
      E/      D822 E100 D822
      FLT     D10590 D824
      FLT     D10593 D826
      E/      D826 E10 D826
; ﾊﾟﾀｰﾝ④実数変換
542   LD      SM400
      AND     M81
      FLT     D10621 D828
      E/      D828 E100 D828
      FLT     D10620 D830
      FLT     D10623 D832
      E/      D832 E10 D832
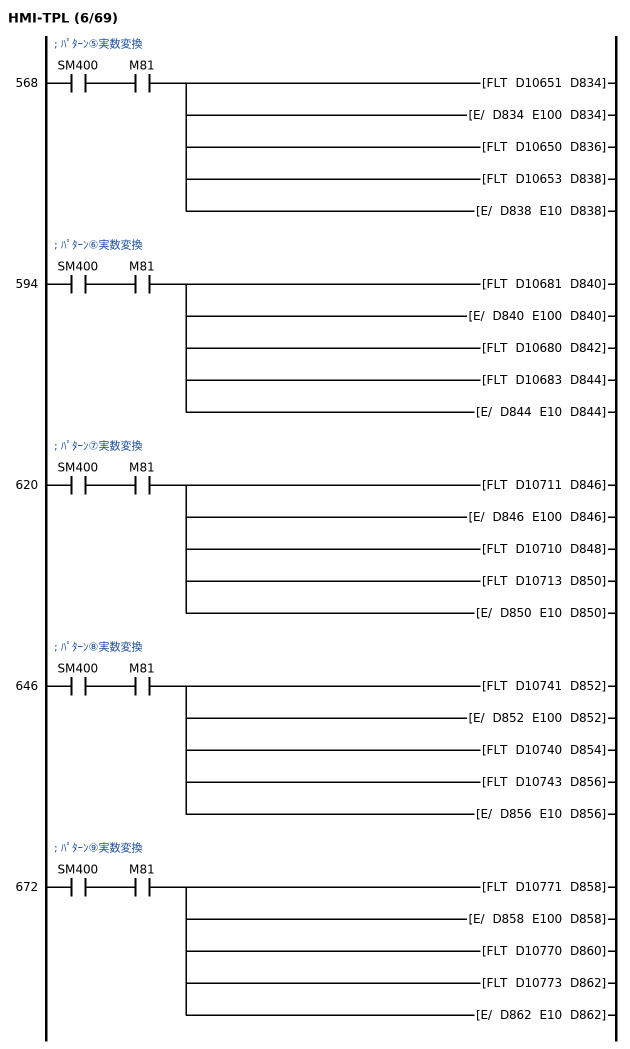
; ﾊﾟﾀｰﾝ⑤実数変換
568   LD      SM400
      AND     M81
      FLT     D10651 D834
      E/      D834 E100 D834
      FLT     D10650 D836
      FLT     D10653 D838
      E/      D838 E10 D838
; ﾊﾟﾀｰﾝ⑥実数変換
594   LD      SM400
      AND     M81
      FLT     D10681 D840
      E/      D840 E100 D840
      FLT     D10680 D842
      FLT     D10683 D844
      E/      D844 E10 D844
; ﾊﾟﾀｰﾝ⑦実数変換
620   LD      SM400
      AND     M81
      FLT     D10711 D846
      E/      D846 E100 D846
      FLT     D10710 D848
      FLT     D10713 D850
      E/      D850 E10 D850
; ﾊﾟﾀｰﾝ⑧実数変換
646   LD      SM400
      AND     M81
      FLT     D10741 D852
      E/      D852 E100 D852
      FLT     D10740 D854
      FLT     D10743 D856
      E/      D856 E10 D856
; ﾊﾟﾀｰﾝ⑨実数変換
672   LD      SM400
      AND     M81
      FLT     D10771 D858
      E/      D858 E100 D858
      FLT     D10770 D860
      FLT     D10773 D862
      E/      D862 E10 D862
